PROGRAM S06_Cutting
VAR
	//工站
	station					: REFERENCE TO FB_Station:=fbstation[6];
	//气缸
	fbGlampCyl_1	:REFERENCE TO FB_Cylinder:=fbCylinder[24];	//	夹膜气缸（前）
	fbGlampCyl_2	:REFERENCE TO FB_Cylinder:=fbCylinder[25];	//	夹膜气缸（后）
	fbHOZReachedCyl_1	:REFERENCE TO FB_Cylinder:=fbCylinder[26];	//	水平到位气缸1
	fbHOZReachedCyl_2	:REFERENCE TO FB_Cylinder:=fbCylinder[27];	//	水平到位气缸2
	fbHOZCyl	:REFERENCE TO FB_Cylinder:=fbCylinder[28];	//	水平切膜气缸
	fbVTCAdjustCyl	:REFERENCE TO FB_Cylinder:=fbCylinder[29];	//	下方顶升调整气缸
	fbGlampAdjustCyl_1	:REFERENCE TO FB_Cylinder:=fbCylinder[30];	//	下方夹爪调整气缸1
	fbGlampAdjustCyl_2	:REFERENCE TO FB_Cylinder:=fbCylinder[31];	//	下方夹爪调整气缸2
	fbGlampAdjustCyl_3	:REFERENCE TO FB_Cylinder:=fbCylinder[32];	//	下方夹爪调整气缸3



	//伺服
	fbROTAxisMove	 :REFERENCE TO FB_Axis:=fbAxis[14];	//	切膜工位丢膜伺服

	//延时
	arTonDelay :ARRAY[1..20] OF TON;
	//返回值
	UdiReturnValue :ARRAY[1..20] OF UDINT;
	//本地过程数据
	arProcessDataStation : ARRAY [1..3] OF DUT_MainlineFixture;
	i: INT;
	// 临时变量
	_FirstCycle:ARRAY[1..10] OF BOOL;
	// 循环计数
	bCounter: BYTE;
	// 结束循环
	bEndCounter: BYTE;
	//过程记录
	tsModuleProcess:ARRAY[1..gc_ModuleProNo] OF DUT_Process;
	xClearModuleProcessDone:BOOL;
	bClearProcessStep	:BYTE;

END_VAR

A_Input();
Alarm();
Delay();
FlowAuto();
FlowInit();
General();
ILC();
TipAuto();
TipManual();
Z_Output();

ACTION A_Input:
//气缸
fbGlampCyl_1.xWP_Sensor	:=	IxS06GlampCyl_1WP AND IxS06GlampCyl_3WP	;
fbGlampCyl_1.xHP_Sensor	:=	IxS06GlampCyl_1HP and IxS06GlampCyl_3HP	;
fbGlampCyl_2.xWP_Sensor	:=	IxS06GlampCyl_2WP and IxS06GlampCyl_4WP	;
fbGlampCyl_2.xHP_Sensor	:=	IxS06GlampCyl_2HP and IxS06GlampCyl_4HP	;
fbHOZReachedCyl_1.xWP_Sensor	:=	IxS06HOZReachedCyl_1WP	;
fbHOZReachedCyl_1.xHP_Sensor	:=	IxS06HOZReachedCyl_1HP	;
fbHOZReachedCyl_2.xWP_Sensor	:=	IxS06HOZReachedCyl_2WP	;
fbHOZReachedCyl_2.xHP_Sensor	:=	IxS06HOZReachedCyl_2HP	;
fbHOZCyl.xWP_Sensor	:=	IxS06HOZCyl_1WP	;
fbHOZCyl.xHP_Sensor	:=	IxS06HOZCyl_1HP	;
fbVTCAdjustCyl.xWP_Sensor	:=	IxS06VTCAdjustCylWP	;
fbVTCAdjustCyl.xHP_Sensor	:=	IxS06VTCAdjustCylHP	;
fbGlampAdjustCyl_1.xWP_Sensor	:=	IxS06GlampAdjustCyl_1WP	;
fbGlampAdjustCyl_1.xHP_Sensor	:=	IxS06GlampAdjustCyl_1HP	;
fbGlampAdjustCyl_2.xWP_Sensor	:=	IxS06GlampAdjustCyl_2WP	;
fbGlampAdjustCyl_2.xHP_Sensor	:=	IxS06GlampAdjustCyl_2HP	;
fbGlampAdjustCyl_3.xWP_Sensor	:=	IxS06GlampAdjustCyl_3WP	;
fbGlampAdjustCyl_3.xHP_Sensor	:=	IxS06GlampAdjustCyl_3HP	;
END_ACTION

ACTION Alarm:
station.adwAlarm[1].00	:=	station.xInitTimeout	;//	S06 初始化超时
station.adwAlarm[1].01	:=	fbGlampCyl_2.xHP_Off	;//	S06切膜工位夹膜气缸(前)原点未到位
station.adwAlarm[1].02	:=	fbGlampCyl_1.xWP_Off	;//	S06切膜工位夹膜气缸(前)动点未到位
station.adwAlarm[1].03	:=	fbGlampCyl_2.xHP_Off	;//	S06切膜工位夹膜气缸(后)原点未到位
station.adwAlarm[1].04	:=	fbGlampCyl_2.xWP_Off	;//	S06切膜工位夹膜气缸(后)动点未到位
station.adwAlarm[1].05	:=	fbHOZReachedCyl_1.xHP_Off 	;//	S06切膜工位水平到位气缸1原点未到位
station.adwAlarm[1].06	:=	fbHOZReachedCyl_1.xWP_Off	;//	S06切膜工位水平到位气缸1动点未到位
station.adwAlarm[1].07	:=	fbHOZReachedCyl_2.xHP_Off	;//	S06切膜工位水平到位气缸2原点未到位
station.adwAlarm[1].08	:=	fbHOZReachedCyl_2.xWP_Off	;//	S06切膜工位水平到位气缸2动点未到位
station.adwAlarm[1].09	:=	fbHOZCyl.xHP_Off 	;//	S06切膜工位水平切膜气缸原点未到位
station.adwAlarm[1].10	:=	fbHOZCyl.xWP_Off 	;//	S06切膜工位水平切膜气缸动点未到位
station.adwAlarm[1].11	:=	fbVTCAdjustCyl.xHP_Off 	;//	S06切膜工位顶升气缸原点未到位
station.adwAlarm[1].12	:=	fbVTCAdjustCyl.xWP_Off 	;//	S06切膜工位顶升气缸动点未到位
station.adwAlarm[1].13	:=	fbGlampAdjustCyl_1.xHP_Off 	;//	S06切膜工位调整夹爪气缸1原点未到位
station.adwAlarm[1].14	:=	fbGlampAdjustCyl_1.xWP_Off	;//	S06切膜工位调整夹爪气缸1动点未到位
station.adwAlarm[1].15	:=	fbGlampAdjustCyl_2.xHP_Off	;//	S06切膜工位调整夹爪气缸2原点未到位
station.adwAlarm[1].16	:=	fbGlampAdjustCyl_2.xWP_Off	;//	S06切膜工位调整夹爪气缸2动点未到位
station.adwAlarm[1].17	:=	fbGlampAdjustCyl_3.xHP_Off	;//	S06切膜工位调整夹爪气缸3原点未到位
station.adwAlarm[1].18	:=	fbGlampAdjustCyl_3.xWP_Off	;//	S06切膜工位调整夹爪气缸3动点未到位
END_ACTION

ACTION Delay:
(*arTonDelay[01](IN:= , PT:=T#0.1S , Q=> , ET=> );*)//TipAuto使用
arTonDelay[02](IN:=  , PT:=T#1S , Q=> , ET=> );
arTonDelay[03](IN:=   , PT:=T#1S , Q=> , ET=> );
arTonDelay[04](IN:= , PT:=T#0.1S , Q=> , ET=> );
arTonDelay[05](IN:= , PT:=T#0.1S , Q=> , ET=> );
arTonDelay[06](IN:= , PT:=T#0.1S , Q=> , ET=> );
arTonDelay[07](IN:= , PT:=T#0.1S , Q=> , ET=> );
arTonDelay[08](IN:= , PT:=T#0.1S , Q=> , ET=> );
arTonDelay[09](IN:= , PT:=T#0.1S , Q=> , ET=> );
END_ACTION

ACTION FlowAuto:

//-----------------------------------------初始化是否完成判断----------------------------------------------
IF NOT station.xInitDone 
THEN
 	station.iStepAuto:=0;
 	station.xDone:=FALSE;
ELSIF station.xRunning OR (  tsModuleProcess[2].xProcessStarted AND   NOT tsModuleProcess[2].xProcessCompleted)
THEN
//-----------------------------------------动作步骤--------------------------------------------------------
CASE station.iStepAuto OF	  
	0: //----Home Step，等待启动----
		IF station.xDisabled 
			AND station.xCanRun 
			AND NOT fbMachine[1].xStopped 
			AND NOT station.xSingleRunning 
		THEN
			station.xDone:=TRUE;
		END_IF
		
		IF  station.xSingleRunning 
			OR station.xCanRun 
			AND NOT station.xDone 
			AND NOT station.xDisabled 
			AND NOT fbMachine[1].xStopped
		THEN
			station.xCycleEnable:=TRUE;
			station.xDone:= FALSE;  
			station.iStepAuto:= 5;
		END_IF
    5: //复位数据 
			//	IF  station.xSingleRunning THEN
				 FOR i:=1 TO gc_ModuleProNo BY 1 DO
						 MEMSET(ADR(tsModuleProcess[i]),0,SIZEOF(tsModuleProcess[i]));
				 END_FOR
		//	END_IF
			station.iStepAuto:=10;
	10: //判断产品是否到该工位
		IF (* fbMachine[1].xTryRun OR*) station.xSingleRunning THEN
			station.iStepAuto:= 20;
		ELSE
			IF   	 NOT  arMainlineFixtureData[arCurFixtureNumStation[14]].xMaterialOnOff AND
					 NOT arMainlineFixtureData[arCurFixtureNumStation[15]].xMaterialOnOff AND 
					 NOT arMainlineFixtureData[arCurFixtureNumStation[16]].xMaterialOnOff THEN
					 xS05WorkPermit:=TRUE;
					station.iStepAuto:= 999;			
			ELSIF	arMainlineFixtureData[arCurFixtureNumStation[14]].xMaterialOnOff AND    
				    arMainlineFixtureData[arCurFixtureNumStation[15]].xMaterialOnOff  AND 
					NOT arMainlineFixtureData[arCurFixtureNumStation[16]].xMaterialOnOff THEN
					station.iStepAuto:= 20;
			ELSIF	NOT arMainlineFixtureData[arCurFixtureNumStation[14]].xMaterialOnOff AND    
				    arMainlineFixtureData[arCurFixtureNumStation[15]].xMaterialOnOff  AND 
					 arMainlineFixtureData[arCurFixtureNumStation[16]].xMaterialOnOff THEN
					station.iStepAuto:= 20;
			END_IF
		END_IF
	20:////Restore_after_Estop_Process1 上载数据流程
			IF  station.xSingleRunning  THEN //OR  fbMachine[1].xTryRun THEN
					station.iStepAuto :=40; 
			ELSIF tsModuleProcess[1].xProcessNotStarted AND NOT  tsModuleProcess[1].xProcessStarted THEN
					station.iStepAuto :=21; (*process not started*)
			ELSIF  tsModuleProcess[1].xProcessStarted AND NOT  tsModuleProcess[1].xProcessCompleted THEN
				 station.iStepAuto := 21;(*process started*)
			ELSIF  tsModuleProcess[1].xProcessCompleted AND NOT tsModuleProcess[1].xQDataCompleted  THEN
					station.iStepAuto := 40 ;(*process completed*)
			ELSIF tsModuleProcess[1].xQDataCompleted THEN
					station.iStepAuto :=40;(*Qdata completed *)
			ELSE
					station.iStepAuto :=21; 
			END_IF	
	21://
				tsModuleProcess[1].xProcessNotStarted:=TRUE;
				station.iStepAuto:= 30;
	30://上载产品数据
			tsModuleProcess[1].xProcessStarted	:=TRUE;
			IF  arMainlineFixtureData[arCurFixtureNumStation[14]].xMaterialOnOff  THEN
				MEMCPY(ADR(arProcessDataStation[1]),ADR(arMainlineFixtureData[arCurFixtureNumStation[14]]),SIZEOF(arMainlineFixtureData[arCurFixtureNumStation[14]]));
			END_IF
				MEMCPY(ADR(arProcessDataStation[2]),ADR(arMainlineFixtureData[arCurFixtureNumStation[15]]),SIZEOF(arMainlineFixtureData[arCurFixtureNumStation[15]]));
			IF  arMainlineFixtureData[arCurFixtureNumStation[16]].xMaterialOnOff THEN
				MEMCPY(ADR(arProcessDataStation[3]),ADR(arMainlineFixtureData[arCurFixtureNumStation[16]]),SIZEOF(arMainlineFixtureData[arCurFixtureNumStation[16]]));
			END_IF
			tsModuleProcess[1].xProcessCompleted:=TRUE;
			station.iStepAuto:= 40;			
	/////产品流程开始	
	40:
		station.iStepAuto:= 50;
	50://下方顶升气缸伸出
		fbVTCAdjustCyl.xAuto:=TRUE;
		IF fbVTCAdjustCyl.xWP_Delay THEN
			station.iStepAuto :=60;	
		END_IF	
	60://下方夹爪气缸夹紧
			IF  arProcessDataStation[1].xMaterialOnOff THEN
				fbGlampAdjustCyl_1.xAuto:=TRUE;
			END_IF
				fbGlampAdjustCyl_2.xAuto:=TRUE;
			IF   arProcessDataStation[3].xMaterialOnOff THEN
				fbGlampAdjustCyl_3.xAuto:=TRUE;
			END_IF
			IF    ( fbGlampAdjustCyl_1.xWP_Delay OR arProcessDataStation[1].xMaterialOnOff=FALSE) AND
				  fbGlampAdjustCyl_2.xWP_Delay  AND 
				  (fbGlampAdjustCyl_3.xWP_Delay OR  arProcessDataStation[3].xMaterialOnOff =FALSE)  THEN
					station.iStepAuto :=65;	
			END_IF
	65://允许调整工位动作
			xS05WorkPermit:=TRUE;
			station.iStepAuto :=70;	
	70://水平到位气缸伸出
		fbHOZReachedCyl_1.xauto :=TRUE;
		fbHOZReachedCyl_2.xauto :=true;
		IF	fbHOZReachedCyl_1.xWP_Delay AND 
			fbHOZReachedCyl_2.xWP_Delay THEN
				station.iStepAuto :=80;	
		END_IF
	80://前后侧夹爪气缸夹住铝膜
		fbGlampCyl_1.xauto :=TRUE;
		fbGlampCyl_2.xauto:=TRUE;
		IF	fbGlampCyl_1.xWP_Delay AND 
			fbGlampCyl_2.xWP_Delay THEN
				station.iStepAuto :=90;	
		END_IF
	90:////Restore_after_Estop_Process2 切膜流程
			IF  station.xSingleRunning OR fbMachine[1].xTryRun THEN
					station.iStepAuto :=100; 
			ELSIF tsModuleProcess[2].xProcessNotStarted AND NOT  tsModuleProcess[2].xProcessStarted THEN
					station.iStepAuto :=110; (*process not started*)
			ELSIF  tsModuleProcess[2].xProcessStarted AND NOT  tsModuleProcess[2].xProcessCompleted THEN
				 station.iStepAuto := 110;(*process started*)
			ELSIF  tsModuleProcess[2].xProcessCompleted AND NOT tsModuleProcess[2].xQDataCompleted  THEN
					station.iStepAuto :=120;(*process completed*)
			ELSIF tsModuleProcess[2].xQDataCompleted THEN
					station.iStepAuto :=130;(*Qdata completed *)
			ELSE
					station.iStepAuto :=100; 
			END_IF	
	100://	
			 tsModuleProcess[2].xProcessNotStarted:=TRUE;
			 station.iStepAuto :=110; 
	
	110://切膜流程开始
			tsModuleProcess[2].xProcessStarted:=TRUE;
			fbHOZCyl.xAuto:=TRUE;
			IF  fbHOZCyl.xWP_Delay THEN
				station.iStepAuto :=120;		
			END_IF
	120:
			tsModuleProcess[2].xProcessCompleted:=TRUE;
			station.iStepAuto :=125;	
	125:	
		IF  arProcessDataStation[1].xMaterialOnOff  THEN
			arProcessDataStation[1].stProduct.xCutting_NOK:=FALSE;
			arProcessDataStation[1].stProduct.xCutting_OK:=TRUE;		
		END_IF
		
		arProcessDataStation[2].stProduct.xCutting_NOK:=FALSE;
		arProcessDataStation[2].stProduct.xCutting_OK:=TRUE;
		
		IF  arProcessDataStation[3].xMaterialOnOff  THEN
			arProcessDataStation[3].stProduct.xCutting_NOK:=FALSE;
			arProcessDataStation[3].stProduct.xCutting_OK:=TRUE;		
		END_IF
		tsModuleProcess[2].xQDataCompleted:=TRUE;
		station.iStepAuto :=130;	
	
	130://后侧夹爪气缸松开
			fbGlampCyl_2.xauto:=FALSE;
			IF	fbGlampCyl_2.xHP_Delay THEN
					station.iStepAuto :=140;	
			END_IF
	140://水平到位气缸收回
			fbHOZReachedCyl_1.xauto :=FALSE;
			fbHOZReachedCyl_2.xauto :=FALSE;
			IF	fbHOZReachedCyl_1.xHP_Delay AND 
				fbHOZReachedCyl_2.xHP_Delay THEN
					station.iStepAuto :=150;	
			END_IF	
	150://旋转伺服去工作位置
		 fbROTAxisMove.xMoveAuto[2]:=TRUE;
		 IF fbROTAxisMove.xMoveInPos[2] THEN
			 station.iStepAuto :=160; 
		 END_IF
	160://水平切膜气缸返回
		 	fbHOZCyl.xAuto:=FALSE;
			IF  fbHOZCyl.xHP_Delay THEN
				station.iStepAuto :=170;		
			END_IF 
	170://调整夹爪气缸松开
				
				fbGlampAdjustCyl_1.xAuto:=FALSE;
				fbGlampAdjustCyl_2.xAuto:=FALSE;
				fbGlampAdjustCyl_3.xAuto:=FALSE;
			IF   fbGlampAdjustCyl_1.xHP_Delay AND
				  fbGlampAdjustCyl_2.xHP_Delay  AND 
				  fbGlampAdjustCyl_3.xHP_Delay   THEN
					station.iStepAuto :=180;	
			END_IF
	180://顶升调整气缸收回
				fbVTCAdjustCyl.xAuto:=FALSE;
		IF fbVTCAdjustCyl.xHP_Delay THEN
			station.iStepAuto :=200;	
		END_IF	
			
	////产品流程结束	
	200:////Restore_after_Estop_Process3 数据传输流程
			IF  station.xSingleRunning THEN // OR fbMachine[1].xTryRun THEN
					station.iStepAuto :=250;
			ELSIF tsModuleProcess[3].xProcessNotStarted AND NOT  tsModuleProcess[3].xProcessStarted THEN
					station.iStepAuto :=210; (*process not started*)
			ELSIF  tsModuleProcess[3].xProcessStarted AND NOT  tsModuleProcess[3].xProcessCompleted THEN
				 station.iStepAuto := 220;(*process started*)
			ELSIF  tsModuleProcess[3].xProcessCompleted AND NOT tsModuleProcess[3].xQDataCompleted  THEN
					station.iStepAuto :=230;(*process completed*)
			ELSIF tsModuleProcess[3].xQDataCompleted THEN
					station.iStepAuto :=250;(*Qdata completed *)
			ELSE
					station.iStepAuto :=210; 
			END_IF		
	210://		
				tsModuleProcess[3].xProcessNotStarted:=TRUE;
				station.iStepAuto :=220; 
	220://数据unload
		tsModuleProcess[3].xProcessStarted:=TRUE;
		IF arProcessDataStation[1].xMaterialOnOff  THEN
			MEMCPY(ADR(arMainlineFixtureData[arCurFixtureNumStation[14]]),ADR(arProcessDataStation[1]),SIZEOF(arProcessDataStation[1]));
		END_IF
		MEMCPY(ADR(arMainlineFixtureData[arCurFixtureNumStation[15]]),ADR(arProcessDataStation[2]),SIZEOF(arProcessDataStation[2]));
		IF arProcessDataStation[3].xMaterialOnOff  THEN
			MEMCPY(ADR(arMainlineFixtureData[arCurFixtureNumStation[16]]),ADR(arProcessDataStation[3]),SIZEOF(arProcessDataStation[3]));
		END_IF
		station.iStepAuto:= 230;
	230://
			tsModuleProcess[3].xProcessCompleted:=TRUE;
			station.iStepAuto :=240; 
 	240://本地数据清除
	//		MEMSET(ADR(arProcessDataStation[1]),0,SIZEOF(arProcessDataStation[1]));
	//		MEMSET(ADR(arProcessDataStation[2]),0,SIZEOF(arProcessDataStation[2]));
	//		MEMSET(ADR(arProcessDataStation[3]),0,SIZEOF(arProcessDataStation[3]));
	//		tsModuleProcess[3].xQDataCompleted:=TRUE;
			station.iStepAuto:= 250;
	250://
				station.xDone:=TRUE;
				station.iStepAuto:= 260;
				
	260://夹爪松开			
			fbGlampCyl_1.xauto:=FALSE;
			IF	fbGlampCyl_1.xHP_Delay THEN
					station.iStepAuto :=270;	
			END_IF
	270://伺服回初始位置		
			fbROTAxisMove.xMoveAuto[1]:=TRUE;
		 IF fbROTAxisMove.xMoveInPos[1] THEN
			 station.iStepAuto :=999; 
		 END_IF
	999://----Single Run Finish----
			
		station.iStepAuto :=0;
		IF NOT station.xSingleContinuousRun THEN
			station.xSingleRunFlag:=FALSE;
		END_IF
		
		station.xCycleEnable:=FALSE;	
		station.xDone:=TRUE;			
		
	ELSE
		;	
END_CASE



END_IF
END_ACTION

ACTION FlowInit:
IF NOT station.xIniting THEN
  station.iStepInit:=0;    
ELSE
//--------------------------------------------初始化步序----------------------------------
CASE station.iStepInit OF	
 0://  
  	IF station.xIniting THEN	
  	  station.iStepInit:=10;	
  	END_IF	
10://复位数据
	FOR i:=1 TO gc_ModuleProNo BY 1 DO
				MEMSET(ADR(tsModuleProcess[i]),0,SIZEOF(tsModuleProcess[i]));
	END_FOR
	station.iStepInit :=40;

//20://切膜流程分析
//		IF   tsModuleProcess[2].xProcessStarted  AND  NOT tsModuleProcess[2].xProcessCompleted  THEN
//			station.iStepInit:=40;
//		ELSIF     tsModuleProcess[2].xProcessCompleted  THEN
//			station.iStepInit:=50;
//		ELSE(*未开始*)
//			station.iStepInit :=200;
//		END_IF

40://水平切膜气缸伸出
	fbHOZCyl.xInit :=TRUE;
	IF  fbHOZCyl.xHP_Delay THEN
		station.iStepInit :=50;
	END_IF
50://后侧夹爪气缸松开
	fbGlampCyl_2.xInit :=TRUE;
	IF   fbGlampCyl_2.xHP_Delay THEN
		station.iStepInit :=60;
	END_IF
60://水平对顶气缸收回
	fbHOZReachedCyl_1.xInit :=TRUE;
	fbHOZReachedCyl_2.xInit :=TRUE;
	IF   fbHOZReachedCyl_1.xHP_Delay AND
		 fbHOZReachedCyl_2.xHP_Delay THEN
		station.iStepInit :=70;
	END_IF	
70:	//旋转伺服上电
	fbROTAxisMove.xPowerInit:=TRUE;
	IF  fbROTAxisMove.xPowerOn THEN
		station.iStepInit :=80;
	END_IF
80://旋转伺服旋转到位置1
	fbROTAxisMove.xMoveAuto[2]:=TRUE;
	IF  fbROTAxisMove.xMoveInPos[2] THEN
		station.iStepInit :=90;
	END_IF
90://水平切莫气缸收回
	fbHOZCyl.xInit:=TRUE;
	IF  fbHOZCyl.xHP_Delay THEN
			station.iStepInit :=100;
	END_IF
	
100://前测夹爪气缸松开
	fbGlampCyl_1.xInit :=TRUE;
	IF   fbGlampCyl_1.xHP_Delay THEN
		station.iStepInit :=250;
	END_IF
(*************流程未开始*****************)
200://水平切膜收回
	fbHOZCyl.xInit:=TRUE;
	IF  fbHOZCyl.xHP_Delay THEN
			station.iStepInit :=210;
	END_IF
210://前后夹爪气缸松开
	fbGlampCyl_1.xInit :=TRUE;
	fbGlampCyl_2.xInit :=TRUE;
	IF   fbGlampCyl_1.xHP_Delay AND
		  fbGlampCyl_2.xHP_Delay THEN
		station.iStepInit :=220;
	END_IF	
220://水平对位气缸收回
	fbHOZReachedCyl_1.xInit :=TRUE;
	fbHOZReachedCyl_2.xInit :=TRUE;
	IF   fbHOZReachedCyl_1.xHP_Delay AND 
		 fbHOZReachedCyl_2.xHP_Delay THEN
		station.iStepInit :=250;
	END_IF	

250://旋转伺服回参考位置
	fbROTAxisMove.xMoveAuto[1]:=TRUE;
	IF  fbROTAxisMove.xMoveInPos[1] THEN
		station.iStepInit :=260;
	END_IF
260://下方夹气缸松开
	fbGlampAdjustCyl_1.xinit :=TRUE;
    fbGlampAdjustCyl_2.xinit :=true;
    fbGlampAdjustCyl_3.xinit :=TRUE;
	IF fbGlampAdjustCyl_1.xHP_Delay AND 
		fbGlampAdjustCyl_2.xHP_Delay AND 
	   fbGlampAdjustCyl_3.xHP_Delay THEN
	   station.iStepInit :=270;	
	END_IF
270://下方顶升气缸回原位
	fbVTCAdjustCyl.xInit:=TRUE;
	IF fbVTCAdjustCyl.xHP_Delay THEN
		station.iStepInit :=300;	
	END_IF
	
300://	
    station.iStepInit:=999;	
999://初始化完成	
	station.iStepInit:=0;
	station.xInitDone:=TRUE;  
END_CASE
END_IF
END_ACTION

ACTION General:
(******************清除过程记录**********************)
CASE bClearProcessStep OF
	0:	
		IF	 S08_MainLine.xClearProcessStatus THEN
			FOR i:=1 TO gc_ModuleProNo BY 1 DO
				MEMSET(ADR(tsModuleProcess[i]),0,SIZEOF(tsModuleProcess[i]));
			END_FOR
			bClearProcessStep:=10;
		END_IF
	10:
		xClearModuleProcessDone:=TRUE;
		bClearProcessStep:=20;
	20:
		IF NOT S08_MainLine.xClearProcessStatus THEN
			xClearModuleProcessDone:=FALSE;
			bClearProcessStep:=30;
		END_IF
	30:  
			bClearProcessStep:=0;
	
END_CASE
END_ACTION

ACTION ILC:

//---------------------------------------------------工站可执行-------------------------------------------------------
station.xCanRun :=TRUE ;

//---------------------------------------------------气缸动作条件-------------------------------------------
fbGlampCyl_1.xOffILC	:=	TRUE	;
fbGlampCyl_1.xOnILC	:=	TRUE	;
fbGlampCyl_2.xOffILC	:=	TRUE	;
fbGlampCyl_2.xOnILC	:=	TRUE	;
fbHOZReachedCyl_1.xOffILC	:=	TRUE	;
fbHOZReachedCyl_1.xOnILC	:=	TRUE	;
fbHOZReachedCyl_2.xOffILC	:=	TRUE	;
fbHOZReachedCyl_2.xOnILC	:=	TRUE	;
fbHOZCyl.xOffILC	:=	TRUE	;
fbHOZCyl.xOnILC	:=	TRUE	;
fbVTCAdjustCyl.xOffILC	:=	TRUE	;
fbVTCAdjustCyl.xOnILC	:=	TRUE	;
fbGlampAdjustCyl_1.xOffILC	:=	TRUE	;
fbGlampAdjustCyl_1.xOnILC	:=	TRUE	;
fbGlampAdjustCyl_2.xOffILC	:=	TRUE	;
fbGlampAdjustCyl_2.xOnILC	:=	TRUE	;
fbGlampAdjustCyl_3.xOffILC	:=	TRUE	;
fbGlampAdjustCyl_3.xOnILC	:=	TRUE	;


//---------------------------------------------------伺服动作条件-------------------------------------------
fbROTAxisMove.xRunILC := TRUE;
fbROTAxisMove.xMoveILC[1] :=fbHOZReachedCyl_1.xHP_Delay AND fbHOZReachedCyl_2.xHP_Delay ;
END_ACTION

ACTION TipAuto:

//------------------------------------------------AutoTip Cylinder--------------------------------
station.adwAutoTip[1].00	:=	fbGlampCyl_1.xAutoTip	;
station.adwAutoTip[1].01	:=	fbGlampCyl_2.xAutoTip	;
station.adwAutoTip[1].02	:=	fbHOZReachedCyl_1.xAutoTip	;
station.adwAutoTip[1].03	:=	fbHOZReachedCyl_2.xAutoTip	;
station.adwAutoTip[1].04	:=	fbHOZCyl.xAutoTip	;
station.adwAutoTip[1].05	:=	fbVTCAdjustCyl.xAutoTip	;
station.adwAutoTip[1].06	:=	fbGlampAdjustCyl_1.xAutoTip	;
station.adwAutoTip[1].07	:=	fbGlampAdjustCyl_2.xAutoTip	;
station.adwAutoTip[1].08	:=	fbGlampAdjustCyl_3.xAutoTip	;

//------------------------------------------------AutoTip Servo--------------------------------
//**************************************
FOR i:= 1 TO 5 BY 1 DO 
	IF fbROTAxisMove.xMoveAuto[i] THEN
		fbROTAxisMove.iPosNumber := i ;
	END_IF
	
END_FOR


IF  fbMachine[1].xAutoMode AND NOT fbMachine[1].xRunning  THEN
	  arTonDelay[01](IN:=True , PT:=T#1S , Q=> , ET=> );
else
	  arTonDelay[01](IN:=false);
END_IF
IF arTonDelay[1].Q  THEN 
		IF	fbROTAxisMove.iPosNumber=1 	AND NOT fbROTAxisMove.xMoveInPos[1] 	THEN 	station.adwAutoTip[1].10:=TRUE	;	END_IF//轴伺服自动时位置不在位置1
		if	fbROTAxisMove.iPosNumber=2	AND NOT fbROTAxisMove.xMoveInPos[2]	THEN 	station.adwAutoTip[1].11:=TRUE	;	END_IF//轴伺服自动时位置不在位置2
		if	fbROTAxisMove.iPosNumber=3	AND NOT fbROTAxisMove.xMoveInPos[3]	THEN 	station.adwAutoTip[1].12:=TRUE	;	END_IF//轴伺服自动时位置不在位置3
		if	fbROTAxisMove.iPosNumber=4	AND NOT fbROTAxisMove.xMoveInPos[4]	THEN 	station.adwAutoTip[1].13:=TRUE	;	END_IF//轴伺服自动时位置不在位置4
		if	fbROTAxisMove.iPosNumber=5	AND NOT fbROTAxisMove.xMoveInPos[5]	THEN 	station.adwAutoTip[1].14:=TRUE	;	END_IF//轴伺服自动时位置不在位置5
END_IF
END_ACTION

ACTION TipManual:
//--------------------------------------------ManualTip------------------------------------------------------

//-------------------------------------------气缸提示---------------------------------------------------------




/////////////////////////////////////////////////////////////////////////////////////////////////////////////////
END_ACTION

ACTION Z_Output:
(**************************气缸输出********************************)
QxS06GlampCyl_1WP	:=	fbGlampCyl_1.xWP_Valve	;
QxS06GlampCyl_1HP	:=	fbGlampCyl_1.xHP_Valve	;
QxS06GlampCyl_2WP	:=	fbGlampCyl_2.xWP_Valve	;
QxS06GlampCyl_2HP	:=	fbGlampCyl_2.xHP_Valve	;
QxS06HOZReachedCyl_1WP	:=	fbHOZReachedCyl_1.xWP_Valve	;
QxS06HOZReachedCyl_1HP	:=	fbHOZReachedCyl_1.xHP_Valve	;
QxS06HOZReachedCyl_2WP	:=	fbHOZReachedCyl_2.xWP_Valve	;
QxS06HOZReachedCyl_2HP	:=	fbHOZReachedCyl_2.xHP_Valve	;
QxS06HOZCyl_1WP	:=	fbHOZCyl.xWP_Valve	;
QxS06HOZCyl_1HP	:=	fbHOZCyl.xHP_Valve	;
QxS06VTCAdjustCylWP	:=	fbVTCAdjustCyl.xWP_Valve	;
QxS06VTCAdjustCylHP	:=	fbVTCAdjustCyl.xHP_Valve	;
QxS06GlampAdjustCyl_1WP	:=	fbGlampAdjustCyl_1.xWP_Valve	;
QxS06GlampAdjustCyl_1HP	:=	fbGlampAdjustCyl_1.xHP_Valve	;
QxS06GlampAdjustCyl_2WP	:=	fbGlampAdjustCyl_2.xWP_Valve	;
QxS06GlampAdjustCyl_2HP	:=	fbGlampAdjustCyl_2.xHP_Valve	;
QxS06GlampAdjustCyl_3WP	:=	fbGlampAdjustCyl_3.xWP_Valve	;
QxS06GlampAdjustCyl_3HP	:=	fbGlampAdjustCyl_3.xHP_Valve	;
END_ACTION

END_PROGRAM

(* stored: Version 1.1.0.1, ProductVersion 3.1.4024.9
   POU S06_Cutting: Id {6d4ccef2-2932-458e-a1b5-77410c4b114d}, SpecialFunc None
   Action A_Input: Id {ac41a8a8-64d1-4ae2-89c0-59150345259a}
   Action Alarm: Id {9eac2c9f-5d99-4890-b419-9170d6594623}
   Action Delay: Id {2180e573-4097-44e6-ba89-ef43671eb619}
   Action FlowAuto: Id {0cc47db4-1390-453c-91c4-9477e61916fa}
   Action FlowInit: Id {16b45474-a7b8-4b9d-aad7-b9de634cbf7e}
   Action General: Id {10dacf65-3705-42c2-8c19-d5ea7aef8a53}
   Action ILC: Id {e9196247-f785-4762-ac90-42ee6c57d7fa}
   Action TipAuto: Id {7c9261bd-b22f-4983-98c6-3e95c5e046e8}
   Action TipManual: Id {1fb9e554-bd39-443a-b880-c4446b214e48}
   Action Z_Output: Id {aa17aaa6-2300-40d4-bd23-1a1fa3da0bc3} *)
